SUBAPPLICATION Button_IXA_TO_logiBUS_QXA_BG_OPC (* Konvertierung Button IXA zu logiBUS QXA und Background *)
  (* Standard: 61499-2; Description: Copyright (c) 2023 Meisterschulen am Ostbahnhof This program and the accompanying materials are made available under the terms of the Eclipse Public License 2.0 which is available at https://www.eclipse.org/legal/epl-2.0/ SPDX-License-Identifier: EPL-2.0 *)
  (* Version 1.1, 2026-07-20, Franz Höpfinger, Meisterschulen am Ostbahnhof, Background *)
  (* Version 1.0, 2026-01-15, Franz Höpfinger, Meisterschulen am Ostbahnhof, initial API and implementation and/or initial documentation *)
  PACKAGE MyLib::sys;
  IMPORT isobus::UT::Q::const::IDs::ID_NULL;
  IMPORT logiBUS::io::DQ::logiBUS_DO;
  IMPORT logiBUS::io::DQ::logiBUS_DO_S;
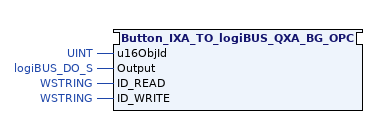
  VAR_INPUT
    u16ObjId : UINT := ID_NULL; (* Object ID *)
    Output : logiBUS::io::DQ::logiBUS_DO_S := logiBUS_DO::Invalid; (* Identify the Output Output_Q1..Q8 *)
    ID_READ : WSTRING;
    ID_WRITE : WSTRING;
  END_VAR
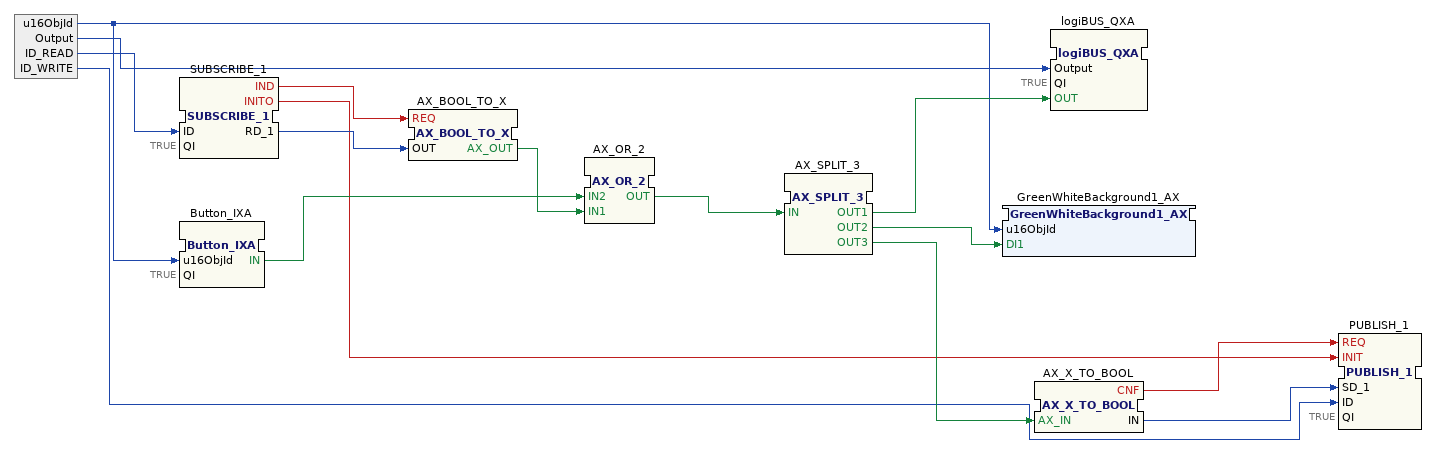
  FBS
    logiBUS_QXA : logiBUS::io::DQ::logiBUS_QXA(QI := TRUE);
    Button_IXA : isobus::UT::io::Button::Button_IXA(QI := TRUE);
    AX_SPLIT_3 : adapter::events::unidirectional::AX_SPLIT_3;
    SUBSCRIBE_1 : iec61499::net::SUBSCRIBE_1(QI := TRUE);
    AX_BOOL_TO_X : adapter::conversion::unidirectional::AX_BOOL_TO_X;
    AX_OR_2 : adapter::booleanOperators::AX_OR_2;
    AX_X_TO_BOOL : adapter::conversion::unidirectional::AX_X_TO_BOOL;
    PUBLISH_1 : iec61499::net::PUBLISH_1(QI := TRUE);
  END_FBS
  SUBAPPS
    GreenWhiteBackground1_AX : MyLib::sys::GreenWhiteBackground1_AX;
  END_SUBAPPS
  EVENT_CONNECTIONS
    SUBSCRIBE_1.IND TO AX_BOOL_TO_X.REQ;
    AX_X_TO_BOOL.CNF TO PUBLISH_1.REQ;
    SUBSCRIBE_1.INITO TO PUBLISH_1.INIT;
  END_CONNECTIONS
  DATA_CONNECTIONS
    u16ObjId TO Button_IXA.u16ObjId;
    Output TO logiBUS_QXA.Output;
    u16ObjId TO GreenWhiteBackground1_AX.u16ObjId;
    ID_READ TO SUBSCRIBE_1.ID;
    SUBSCRIBE_1.RD_1 TO AX_BOOL_TO_X.OUT;
    AX_X_TO_BOOL.IN TO PUBLISH_1.SD_1;
    ID_WRITE TO PUBLISH_1.ID;
  END_CONNECTIONS
  ADAPTER_CONNECTIONS
    Button_IXA.IN TO AX_OR_2.IN2;
    AX_SPLIT_3.OUT1 TO logiBUS_QXA.OUT;
    AX_SPLIT_3.OUT2 TO GreenWhiteBackground1_AX.DI1;
    AX_BOOL_TO_X.AX_OUT TO AX_OR_2.IN1;
    AX_OR_2.OUT TO AX_SPLIT_3.IN;
    AX_SPLIT_3.OUT3 TO AX_X_TO_BOOL.AX_IN;
  END_CONNECTIONS
END_SUBAPPLICATION
